// TwinCAT 3 PLC project PLC_FMS_TEST
// ProgramVersion: 3.1.4024.12
// libraries:
//   Tc2_Standard, * (Beckhoff Automation GmbH)
//   Tc2_System, * (Beckhoff Automation GmbH)
//   Tc3_Module, * (Beckhoff Automation GmbH)
// project tree:
//   GVLs/ GVL_Devices.TcGVL
//   / PlcTask.TcTTO (not stored)
//   POUs/ FB_LeakSensor.TcPOU (not stored), FB_PCWflow.TcPOU (not stored), FB_TempSensor.TcPOU (not stored), FB_TempSensor_2git.TcPOU (not stored), MAIN.TcPOU
// real-time tasks:
//   TASK PlcTask: cycle T#10ms, priority 20, ADS port 350
// I/O:
//   DEVICE Device 1 (EtherCAT), AmsNetId 172.21.42.126.2.1

// ---- GVLs/GVL_Devices.TcGVL
{attribute 'qualified_only'}
VAR_GLOBAL

 {attribute 'pytmc' := '
            pv: FMS:RTD:01
         '}

{attribute 'TcLinkTo' := '.fTemperature := TIIB[Term 1 (EL3208)]^Channel 1^Input;

'}
fbTempSensor1 : FB_TempSensor; //edit if decided to use _2git


{attribute 'pytmc' := '
            pv: FMS:PCW:RTD:01
         '}

{attribute 'TcLinkTo' := '.fTemperature := TIIB[Term 1 (EL3208)]^Channel 1^Input;

'}
fbTempSensor2 : FB_TempSensor; //for PCW temp spot sensor
 

 {attribute 'pytmc' := '
            pv: FMS:LeakSensor:01
         '}

{attribute 'TcLinkTo' := '.fLeakSensor := TIIB[Term 1 (EL1004)]^Channel 1^Input;

'}
fbLeakSensor1 : FB_LeakSensor;

 

 {attribute 'pytmc' := '
            pv: FMS:PCW:01
         '}

{attribute 'TcLinkTo' := '.fPLCflow := TIIB[Term 1 (EL3174)]^Channel 1^Input;

'}
fbPCWflow : FB_PCWflow;

END_VAR

// ---- POUs/MAIN.TcPOU
PROGRAM MAIN
VAR
END_VAR

END_PROGRAM
